TYPE "ValveMachine_Cin"
VERSION : 0.1
// Block: ValveMachine_Cin
   STRUCT
      Manager : ValveMachine_Manager;
      PressureRunning : Bool;
      Rest_ExtEnable : Bool;
      Work_ExtEnable : Bool;
      ExternalAlarms : Bool;
   END_STRUCT;

END_TYPE
